PROGRAM Stn9
VAR

	start9: BOOL;
	reset9: BOOL;

	Stn9ProcessFE: F_TRIG;
	Stn9ProcessRE: R_TRIG;
	bCutStn9ProcessHalt: BOOL;
	DoorClose9: R_TRIG;
	bStn9DoorClamp: BOOL;

END_VAR
VAR // added by the converter: edge detectors and wires of the graphical bodies
    _w1 : BOOL;
    _w2, _w3, _w5, _w6 : ANY;
    _w4 : INT;
END_VAR

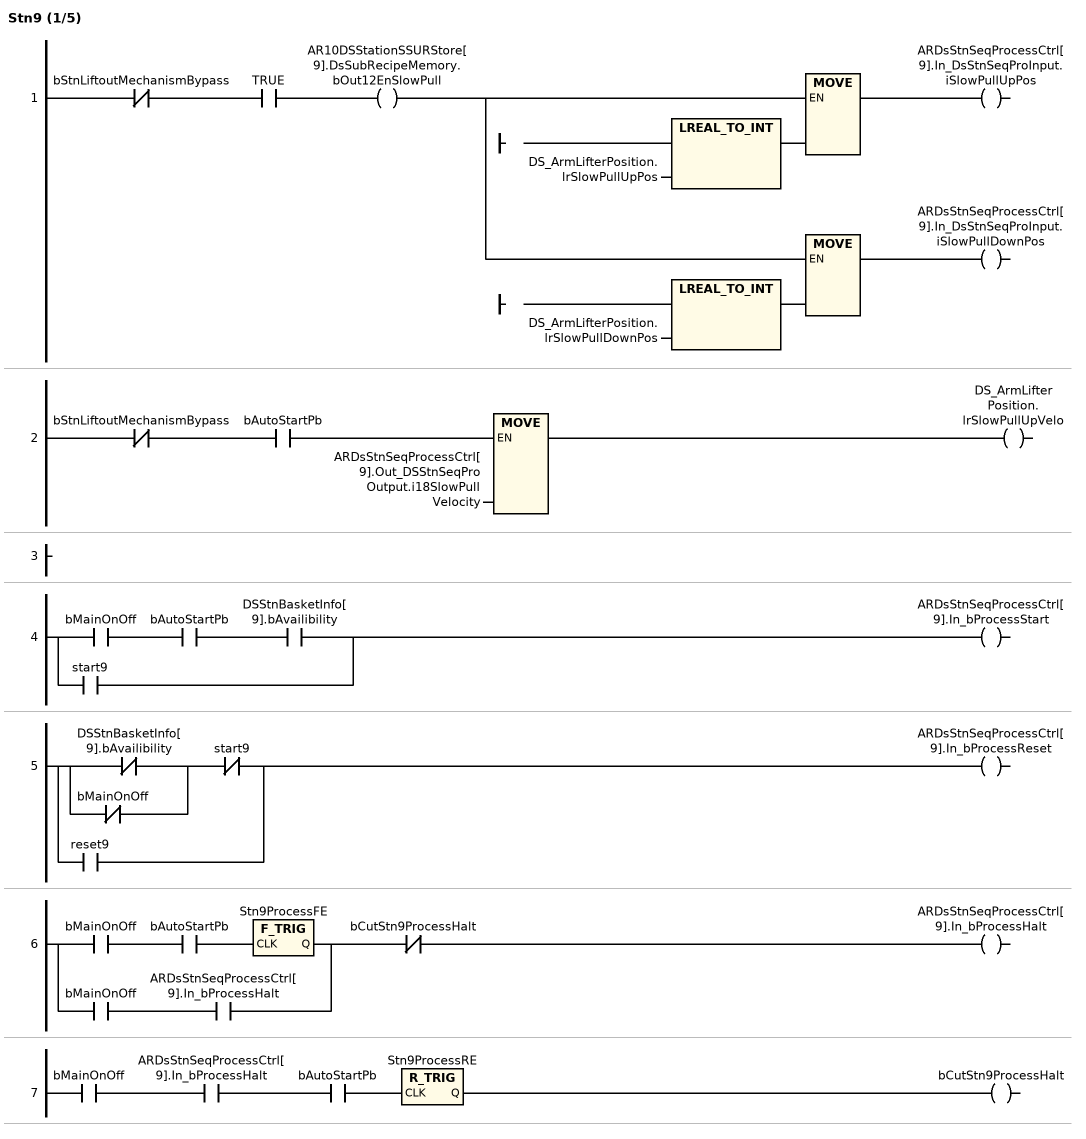
// NETWORK 1
_w1 := NOT bStnLiftoutMechanismBypass AND TRUE;
AR10DSStationSSURStore[9].DsSubRecipeMemory.bOut12EnSlowPull := _w1;
IF _w1 THEN _w2 := LREAL_TO_INT(DS_ArmLifterPosition.lrSlowPullUpPos); END_IF
ARDsStnSeqProcessCtrl[9].In_DsStnSeqProInput.iSlowPullUpPos := _w2;
IF _w1 THEN _w3 := LREAL_TO_INT(DS_ArmLifterPosition.lrSlowPullDownPos); END_IF
ARDsStnSeqProcessCtrl[9].In_DsStnSeqProInput.iSlowPullDownPos := _w3;

// NETWORK 2
IF NOT bStnLiftoutMechanismBypass AND bAutoStartPb THEN
    _w4 := ARDsStnSeqProcessCtrl[9].Out_DSStnSeqProOutput.i18SlowPullVelocity;
END_IF
DS_ArmLifterPosition.lrSlowPullUpVelo := _w4;

// NETWORK 3

// NETWORK 4
ARDsStnSeqProcessCtrl[9].In_bProcessStart := bMainOnOff AND bAutoStartPb AND DSStnBasketInfo[9].bAvailibility OR start9;

// NETWORK 5
ARDsStnSeqProcessCtrl[9].In_bProcessReset := (NOT DSStnBasketInfo[9].bAvailibility OR NOT bMainOnOff) AND NOT start9 OR reset9;

// NETWORK 6
Stn9ProcessFE(CLK := bMainOnOff AND bAutoStartPb); // F_TRIG
ARDsStnSeqProcessCtrl[9].In_bProcessHalt := (Stn9ProcessFE.Q OR bMainOnOff AND ARDsStnSeqProcessCtrl[9].In_bProcessHalt) AND NOT bCutStn9ProcessHalt;

// NETWORK 7
Stn9ProcessRE(CLK := bMainOnOff AND ARDsStnSeqProcessCtrl[9].In_bProcessHalt AND bAutoStartPb); // R_TRIG
bCutStn9ProcessHalt := Stn9ProcessRE.Q;

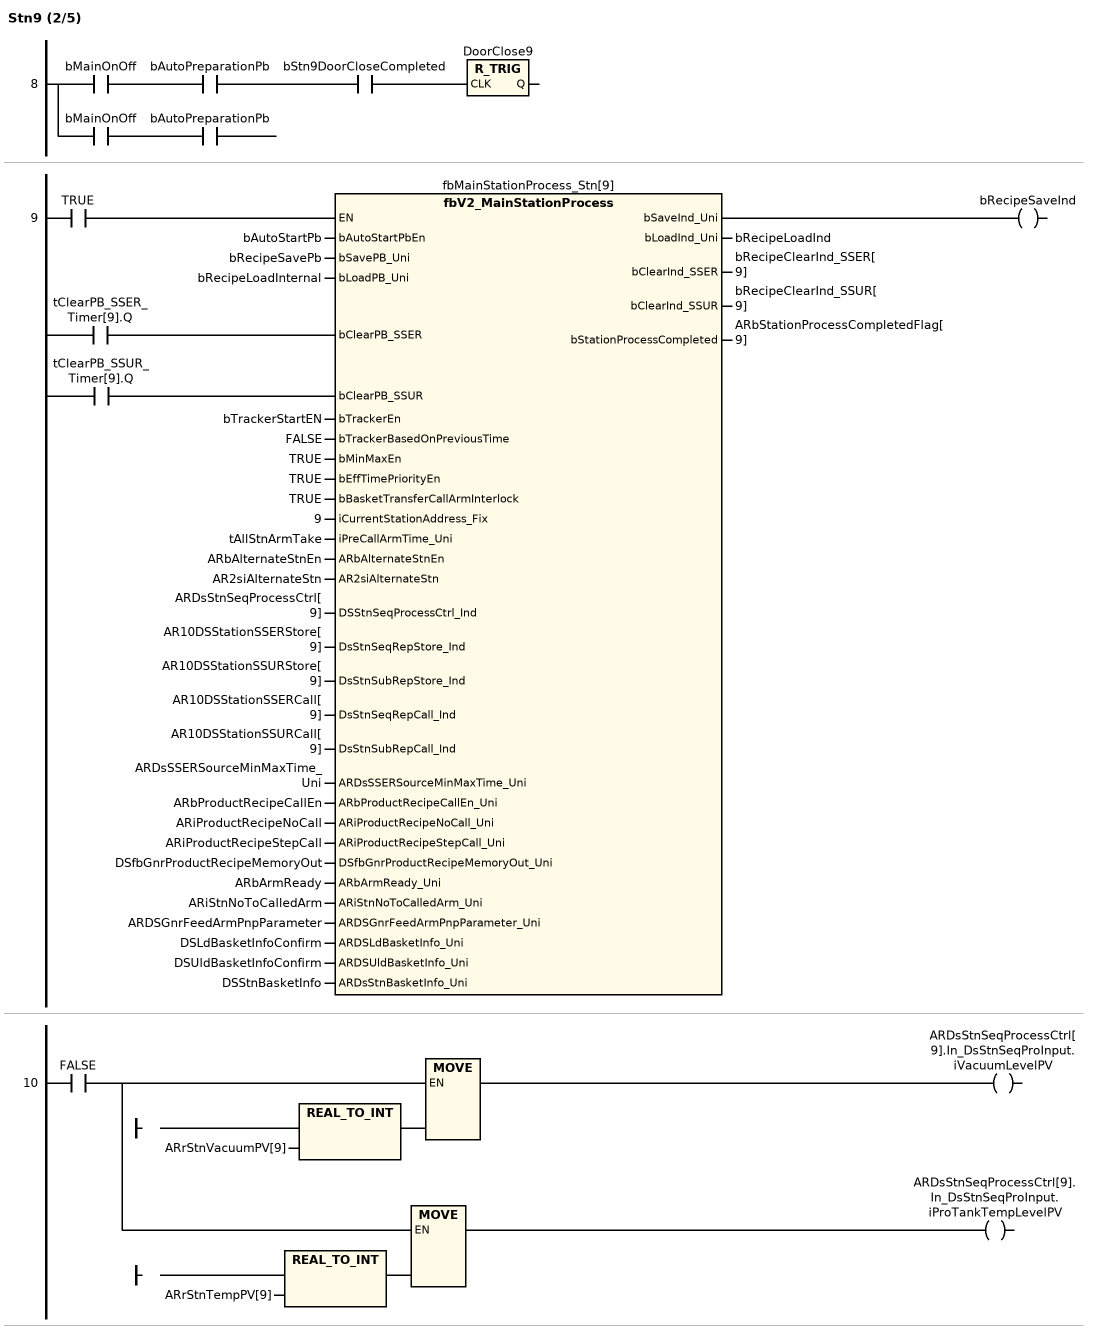
// NETWORK 8
DoorClose9(CLK := bMainOnOff AND bAutoPreparationPb AND bStn9DoorCloseCompleted); // R_TRIG
(* DoorClose9.Q OR bMainOnOff AND bAutoPreparationPb; result not used *)

// NETWORK 9
fbMainStationProcess_Stn[9](
    bAutoStartPbEn := bAutoStartPb,
    bSavePB_Uni := bRecipeSavePb,
    bLoadPB_Uni := bRecipeLoadInternal,
    bClearPB_SSER := tClearPB_SSER_Timer[9].Q,
    bClearPB_SSUR := tClearPB_SSUR_Timer[9].Q,
    bTrackerEn := bTrackerStartEN,
    bTrackerBasedOnPreviousTime := FALSE,
    bMinMaxEn := TRUE,
    bEffTimePriorityEn := TRUE,
    bBasketTransferCallArmInterlock := TRUE,
    iCurrentStationAddress_Fix := 9,
    iPreCallArmTime_Uni := tAllStnArmTake,
    ARbAlternateStnEn := ARbAlternateStnEn,
    AR2siAlternateStn := AR2siAlternateStn,
    DSStnSeqProcessCtrl_Ind := ARDsStnSeqProcessCtrl[9],
    DsStnSeqRepStore_Ind := AR10DSStationSSERStore[9],
    DsStnSubRepStore_Ind := AR10DSStationSSURStore[9],
    DsStnSeqRepCall_Ind := AR10DSStationSSERCall[9],
    DsStnSubRepCall_Ind := AR10DSStationSSURCall[9],
    ARDsSSERSourceMinMaxTime_Uni := ARDsSSERSourceMinMaxTime_Uni,
    ARbProductRecipeCallEn_Uni := ARbProductRecipeCallEn,
    ARiProductRecipeNoCall_Uni := ARiProductRecipeNoCall,
    ARiProductRecipeStepCall_Uni := ARiProductRecipeStepCall,
    DSfbGnrProductRecipeMemoryOut_Uni := DSfbGnrProductRecipeMemoryOut,
    ARbArmReady_Uni := ARbArmReady,
    ARiStnNoToCalledArm_Uni := ARiStnNoToCalledArm,
    ARDSGnrFeedArmPnpParameter_Uni := ARDSGnrFeedArmPnpParameter,
    ARDSLdBasketInfo_Uni := DSLdBasketInfoConfirm,
    ARDSUldBasketInfo_Uni := DSUldBasketInfoConfirm,
    ARDsStnBasketInfo_Uni := DSStnBasketInfo,
    bLoadInd_Uni => bRecipeLoadInd,
    bClearInd_SSER => bRecipeClearInd_SSER[9],
    bClearInd_SSUR => bRecipeClearInd_SSUR[9],
    bStationProcessCompleted => ARbStationProcessCompletedFlag[9]); // fbV2_MainStationProcess
bRecipeSaveInd := fbMainStationProcess_Stn[9].bSaveInd_Uni;

// NETWORK 10
IF FALSE THEN _w5 := REAL_TO_INT(ARrStnVacuumPV[9]); END_IF
ARDsStnSeqProcessCtrl[9].In_DsStnSeqProInput.iVacuumLevelPV := _w5;
IF FALSE THEN _w6 := REAL_TO_INT(ARrStnTempPV[9]); END_IF
ARDsStnSeqProcessCtrl[9].In_DsStnSeqProInput.iProTankTempLevelPV := _w6;

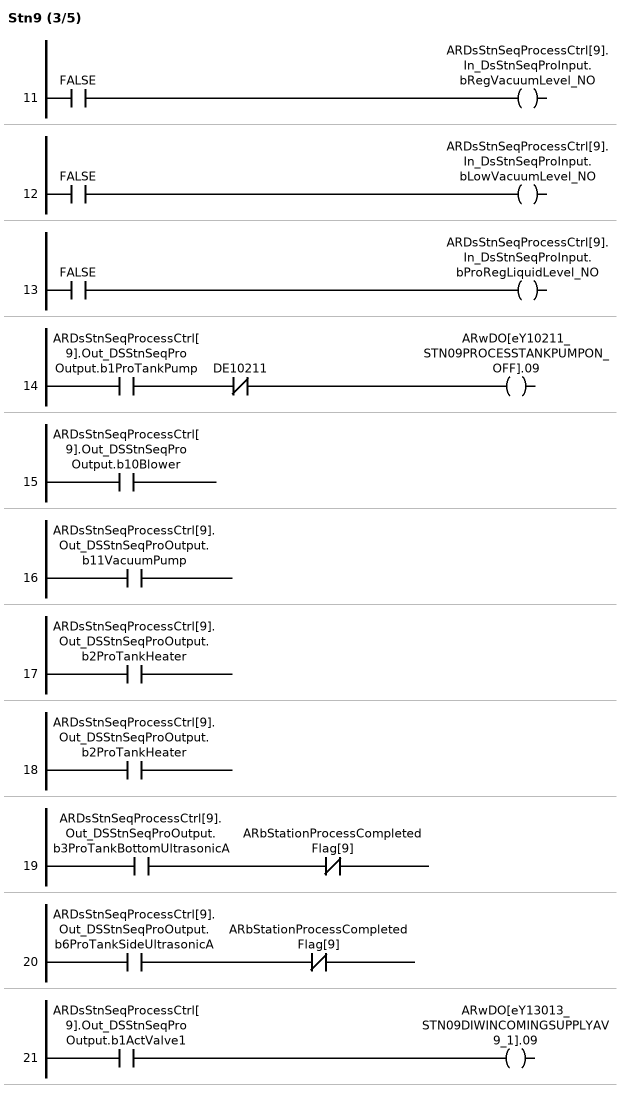
// NETWORK 11
ARDsStnSeqProcessCtrl[9].In_DsStnSeqProInput.bRegVacuumLevel_NO := FALSE;

// NETWORK 12
ARDsStnSeqProcessCtrl[9].In_DsStnSeqProInput.bLowVacuumLevel_NO := FALSE;

// NETWORK 13
ARDsStnSeqProcessCtrl[9].In_DsStnSeqProInput.bProRegLiquidLevel_NO := FALSE;

// NETWORK 14
ARwDO[eY10211_STN09PROCESSTANKPUMPON_OFF].09 := ARDsStnSeqProcessCtrl[9].Out_DSStnSeqProOutput.b1ProTankPump AND NOT DE10211;

// NETWORK 15
(* ARDsStnSeqProcessCtrl[9].Out_DSStnSeqProOutput.b10Blower; not connected *)

// NETWORK 16
(* ARDsStnSeqProcessCtrl[9].Out_DSStnSeqProOutput.b11VacuumPump; not connected *)

// NETWORK 17
(* ARDsStnSeqProcessCtrl[9].Out_DSStnSeqProOutput.b2ProTankHeater; not connected *)

// NETWORK 18
(* ARDsStnSeqProcessCtrl[9].Out_DSStnSeqProOutput.b2ProTankHeater; not connected *)

// NETWORK 19
(* ARDsStnSeqProcessCtrl[9].Out_DSStnSeqProOutput.b3ProTankBottomUltrasonicA AND NOT ARbStationProcessCompletedFlag[9]; result not used *)

// NETWORK 20
(* ARDsStnSeqProcessCtrl[9].Out_DSStnSeqProOutput.b6ProTankSideUltrasonicA AND NOT ARbStationProcessCompletedFlag[9]; result not used *)

// NETWORK 21
ARwDO[eY13013_STN09DIWINCOMINGSUPPLYAV9_1].09 := ARDsStnSeqProcessCtrl[9].Out_DSStnSeqProOutput.b1ActValve1;

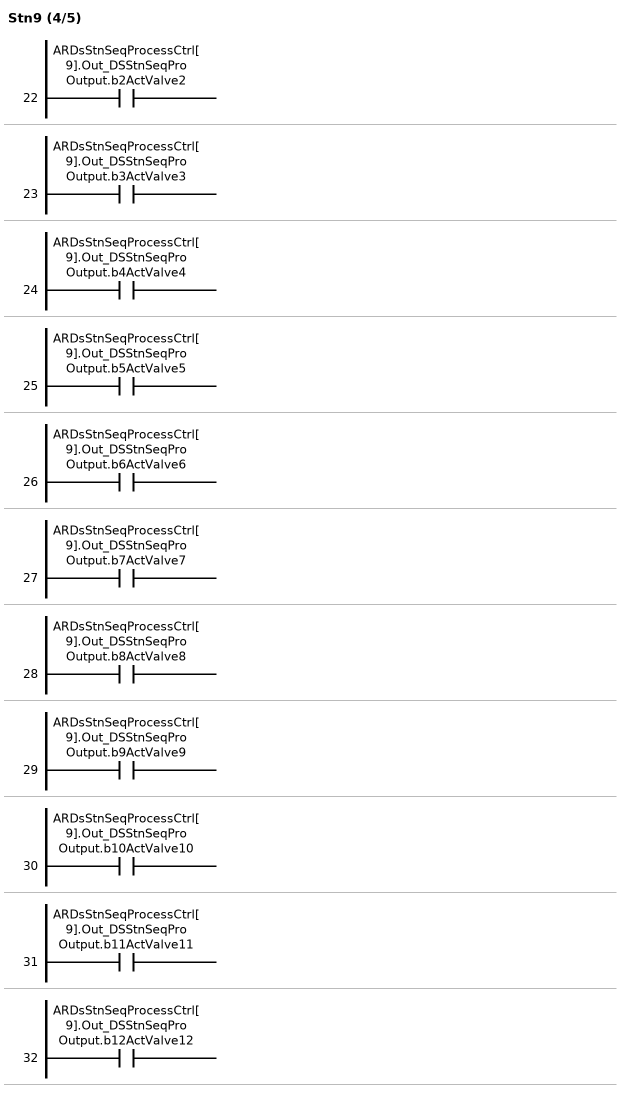
// NETWORK 22
(* ARDsStnSeqProcessCtrl[9].Out_DSStnSeqProOutput.b2ActValve2; not connected *)

// NETWORK 23
(* ARDsStnSeqProcessCtrl[9].Out_DSStnSeqProOutput.b3ActValve3; not connected *)

// NETWORK 24
(* ARDsStnSeqProcessCtrl[9].Out_DSStnSeqProOutput.b4ActValve4; not connected *)

// NETWORK 25
(* ARDsStnSeqProcessCtrl[9].Out_DSStnSeqProOutput.b5ActValve5; not connected *)

// NETWORK 26
(* ARDsStnSeqProcessCtrl[9].Out_DSStnSeqProOutput.b6ActValve6; not connected *)

// NETWORK 27
(* ARDsStnSeqProcessCtrl[9].Out_DSStnSeqProOutput.b7ActValve7; not connected *)

// NETWORK 28
(* ARDsStnSeqProcessCtrl[9].Out_DSStnSeqProOutput.b8ActValve8; not connected *)

// NETWORK 29
(* ARDsStnSeqProcessCtrl[9].Out_DSStnSeqProOutput.b9ActValve9; not connected *)

// NETWORK 30
(* ARDsStnSeqProcessCtrl[9].Out_DSStnSeqProOutput.b10ActValve10; not connected *)

// NETWORK 31
(* ARDsStnSeqProcessCtrl[9].Out_DSStnSeqProOutput.b11ActValve11; not connected *)

// NETWORK 32
(* ARDsStnSeqProcessCtrl[9].Out_DSStnSeqProOutput.b12ActValve12; not connected *)

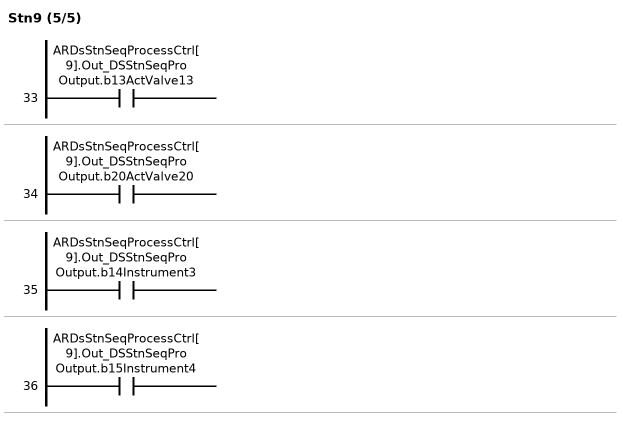
// NETWORK 33
(* ARDsStnSeqProcessCtrl[9].Out_DSStnSeqProOutput.b13ActValve13; not connected *)

// NETWORK 34
(* ARDsStnSeqProcessCtrl[9].Out_DSStnSeqProOutput.b20ActValve20; not connected *)

// NETWORK 35
(* ARDsStnSeqProcessCtrl[9].Out_DSStnSeqProOutput.b14Instrument3; not connected *)

// NETWORK 36
(* ARDsStnSeqProcessCtrl[9].Out_DSStnSeqProOutput.b15Instrument4; not connected *)

END_PROGRAM

(* stored: Version 1.1.0.1, ProductVersion 3.1.4024.12
   POU Stn9: Id {7ce53ae0-6713-4163-9800-e9cb3ef0f550}, SpecialFunc None *)
